FUNCTION_BLOCK FB_ControlE_TE2 EXTENDS FB_BaseControlElement IMPLEMENTS ITF_ControlE_TE2, ITF_ControlE_TE2_HMI_Init
VAR
	itfC1				: ITF_Component_TE2;
	itfC2				: ITF_Component_TE2;
	itfC3				: ITF_Component_TE2;
	itfC4				: ITF_Component_TE2;
	
END_VAR

METHOD FB_init : BOOL
VAR_INPUT
	bInitRetains : BOOL; // if TRUE, the retain variables are initialized (warm start / cold start)
	bInCopyCode : BOOL;  // if TRUE, the instance afterwards gets moved into the copy code (online change)
	itfC1				: ITF_Component_TE2;
	itfC2				: ITF_Component_TE2;
	itfC3				: ITF_Component_TE2;
	itfC4				: ITF_Component_TE2;
END_VAR
THIS^.itfC1 := itfC1;
THIS^.SetText (eLocation := E_BaseLocation.pl, wsDescription := "Komponent 1 EC");
THIS^.SetText (eLocation := E_BaseLocation.en, wsDescription := "Komponent 1 EC");
THIS^.SetText (eLocation := E_BaseLocation.de, wsDescription := "Komponent 1 EC");
itfC1.SetName (stName := THIS^.GetTexts ());
THIS^.AddComponent (itfComponent := itfC1);

THIS^.itfC2 := itfC2;
THIS^.SetText (eLocation := E_BaseLocation.pl, wsDescription := "Komponent 2 EC");
THIS^.SetText (eLocation := E_BaseLocation.en, wsDescription := "Komponent 2 EC");
THIS^.SetText (eLocation := E_BaseLocation.de, wsDescription := "Komponent 2 EC");
itfC2.SetName (stName := THIS^.GetTexts ());
THIS^.AddComponent (itfComponent := itfC2);

THIS^.itfC3 := itfC3;
THIS^.SetText (eLocation := E_BaseLocation.pl, wsDescription := "Komponent 3 EC");
THIS^.SetText (eLocation := E_BaseLocation.en, wsDescription := "Komponent 3 EC");
THIS^.SetText (eLocation := E_BaseLocation.de, wsDescription := "Komponent 3 EC");
itfC3.SetName (stName := THIS^.GetTexts ());
THIS^.AddComponent (itfComponent := itfC3);

THIS^.itfC4 := itfC4;
THIS^.SetText (eLocation := E_BaseLocation.pl, wsDescription := "Komponent 4 EC");
THIS^.SetText (eLocation := E_BaseLocation.en, wsDescription := "Komponent 4 EC");
THIS^.SetText (eLocation := E_BaseLocation.de, wsDescription := "Komponent 4 EC");
itfC4.SetName (stName := THIS^.GetTexts ());
THIS^.AddComponent (itfComponent := itfC4);
END_METHOD

METHOD testMethodCE : BOOL
VAR_INPUT
END_VAR
END_METHOD

END_FUNCTION_BLOCK

(* stored: Version 1.1.0.1, ProductVersion 3.1.4024.15
   POU FB_ControlE_TE2: Id {cdcdcbdb-6505-4a78-ad0c-f177a1b69455}, SpecialFunc None
   Method FB_init: Id {6805b71c-4229-45eb-86b2-e5f37af6302a}
   Method testMethodCE: Id {9287d3df-ab5f-4a44-ad16-ffb35dbb5010} *)
